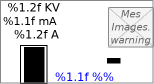
VISUALIZATION VISU_SOURCE_EVAP_COTE_GENIUS_ETH  // 154x84
VAR_IN_OUT
	m_Input_SOURCE : BLOCK_SOURCE_GENIUS_ETHERCAT;
END_VAR
VAR_INPUT
	m_Input_NO_IFIL_RET : BOOL;
	m_Input_NO_HV_RET : BOOL;
	m_Input_NO_IEMISS_RET : BOOL;
END_VAR
    Polygon (84,73), colour toggle: m_Input_SOURCE.STATE_SRC_ON, invisible if: NOT m_Input_SOURCE.STATE_SRC_ON AND NOT m_Input_SOURCE.STATE_SRC
    Polygon (84,71), invisible if: m_Input_SOURCE.STATE_SRC_ON OR (m_Input_SOURCE.STATE_SRC OR m_Input_SOURCE.STATE_SRC)
    Polygon (70,46)
    Polygon (84,43), invisible if: NOT (m_Input_SOURCE.SRC.STATE_On AND m_Input_SOURCE.HV.STATE_On AND (m_Input_SOURCE.STATE_I_EMISS>0.0))
    Rectangle (1,15 62x13), "%1.1f mA", text variable: m_Input_SOURCE.STATE_I_EMISS, invisible if: m_Input_NO_IEMISS_RET
    Rectangle (45,70 79x14), "%1.1f %%", text variable: m_Input_SOURCE.STATE_COURANT
    Rectangle (47,46 77x37), invisible if: (NOT m_Input_SOURCE.SRC.AUTOR_ON_IHM AND NOT m_Input_SOURCE.SRC.AUTOR_OFF_IHM) OR NOT PRG_User.ACTU_USER.MAINTENANCE, input disabled if: (NOT m_Input_SOURCE.SRC.AUTOR_ON_IHM AND NOT m_Input_SOURCE.SRC.AUTOR_OFF_IHM) OR NOT PRG_User.ACTU_USER.MAINTENANCE
        OnMouseUp: execute { m_Input_SOURCE.SRC.M_On:=(TRUE); }
    Rectangle (107,58 13x5), colour toggle: m_Input_SOURCE.WATER
    Rectangle (3,28 59x13), "%1.2f A", text variable: m_Input_SOURCE.STATE_I_Fil, invisible if: m_Input_NO_IFIL_RET
    Image (108,7 46x40), invisible if: NOT m_Input_SOURCE.STATE_NOK, image: MesImages.warning
    Rectangle (1,1 62x13), "%1.2f KV", text variable: m_Input_SOURCE.STATE_V_HV, invisible if: m_Input_NO_HV_RET
    Rectangle (24,47 20x34), colour toggle: (m_Input_SOURCE.STATE_HV_ON), invisible if: NOT m_Input_SOURCE.STATE_HV_ON AND NOT m_Input_SOURCE.STATE_HV
    Rectangle (24,47 20x35), invisible if: (m_Input_SOURCE.STATE_HV_ON OR m_Input_SOURCE.STATE_HV)
    Polygon (41,73)
    Rectangle (20,45 27x39), invisible if: NOT m_Input_SOURCE.HV.AUTOR_ON_IHM AND NOT m_Input_SOURCE.HV.AUTOR_OFF_IHM, input disabled if: (NOT m_Input_SOURCE.HV.AUTOR_ON_IHM AND NOT m_Input_SOURCE.HV.AUTOR_OFF_IHM) OR NOT PRG_User.ACTU_USER.MAINTENANCE
        OnMouseUp: execute { m_Input_SOURCE.HV.M_On:=(TRUE); }
END_VISUALIZATION

(* stored: Version 1.1.0.1, ProductVersion 3.1.4024.10
   Visu VISU_SOURCE_EVAP_COTE_GENIUS_ETH: Id {5e515887-e780-4818-a5d8-5e6f9a938c76} *)
